Omron CX-Programmer project NewProject (CX-Programmer 9.73)

# PLC NewPLC1: CP1L M

## Global symbols (name address type ; comment)
0.00 BOOL  ; START
0.01 BOOL  ; STOP
0.02 BOOL  ; SOL 2A
0.03 BOOL  ; SOL 2B
0.04 BOOL  ; SOL 3A
0.05 BOOL  ; SOL 4A
0.06 BOOL  ; CONVEYOR
0.07 BOOL  ; RODLESS L
0.08 BOOL  ; RODLESS R
0.10 BOOL  ; GRIPPER CLOSE
0.11 BOOL  ; 3A UP
100.00 BOOL  ; 1A
100.01 BOOL  ; 1B
100.02 BOOL  ; SOL 2A
100.03 BOOL  ; SOL 2B
100.04 BOOL  ; SOL 3A
100.05 BOOL  ; SOL 4A
100.06 BOOL  ; CONVEYOR
1.00 BOOL  ; 3A DOWN
200.00 BOOL  ; TRIGGER
200.01 BOOL  ; 3A UP
200.02 BOOL  ; 3A DOWN
200.03 BOOL  ; 4A OPEN
200.04 BOOL  ; RESET 3A
200.05 BOOL  ; OFF 1B ON 1A
200.06 BOOL  ; RESET
200.07 BOOL  ; RELAY2
200.10 BOOL  ; RELAY3
200.11 BOOL  ; RELAY4
300.00 BOOL  ; RELAY1

## Program UT2 (cyclic task 0)

### Section Section1

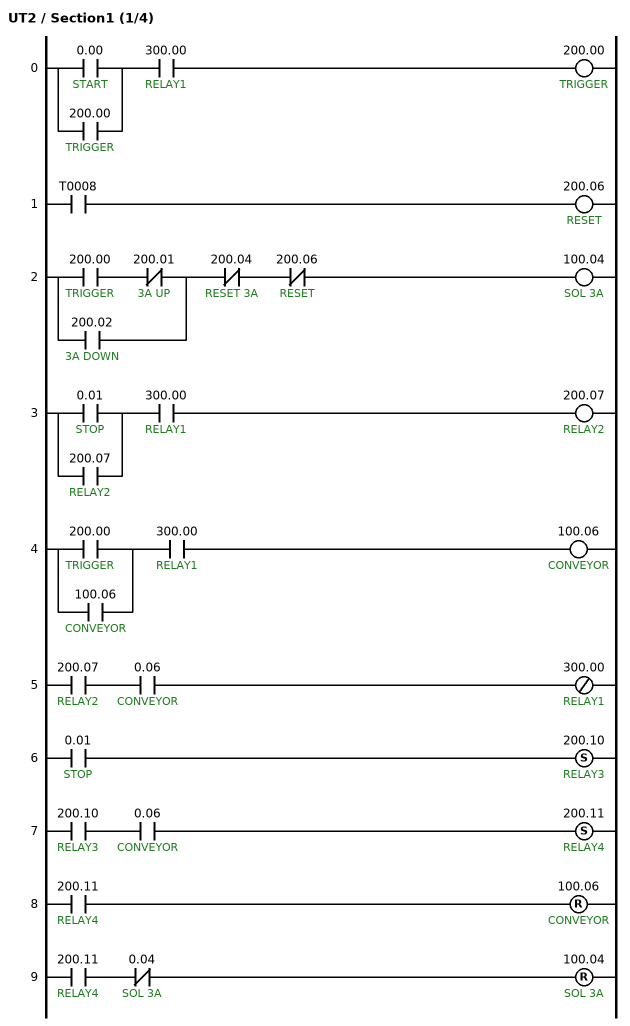
; rung 0
LD 0.00  ; START
OR 200.00  ; TRIGGER
AND 300.00  ; RELAY1
OUT 200.00  ; TRIGGER
; rung 1
LD T0008
OUT 200.06  ; RESET
; rung 2
LD 200.00  ; TRIGGER
ANDNOT 200.01  ; 3A UP
OR 200.02  ; 3A DOWN
ANDNOT 200.04  ; RESET 3A
ANDNOT 200.06  ; RESET
OUT 100.04  ; SOL 3A
; rung 3
LD 0.01  ; STOP
OR 200.07  ; RELAY2
AND 300.00  ; RELAY1
OUT 200.07  ; RELAY2
; rung 4
LD 200.00  ; TRIGGER
OR 100.06  ; CONVEYOR
AND 300.00  ; RELAY1
OUT 100.06  ; CONVEYOR
; rung 5
LD 200.07  ; RELAY2
AND 0.06  ; CONVEYOR
OUTNOT 300.00  ; RELAY1
; rung 6
LD 0.01  ; STOP
SET 200.10  ; RELAY3
; rung 7
LD 200.10  ; RELAY3
AND 0.06  ; CONVEYOR
SET 200.11  ; RELAY4
; rung 8
LD 200.11  ; RELAY4
RSET 100.06  ; CONVEYOR
; rung 9
LD 200.11  ; RELAY4
ANDNOT 0.04  ; SOL 3A
RSET 100.04  ; SOL 3A

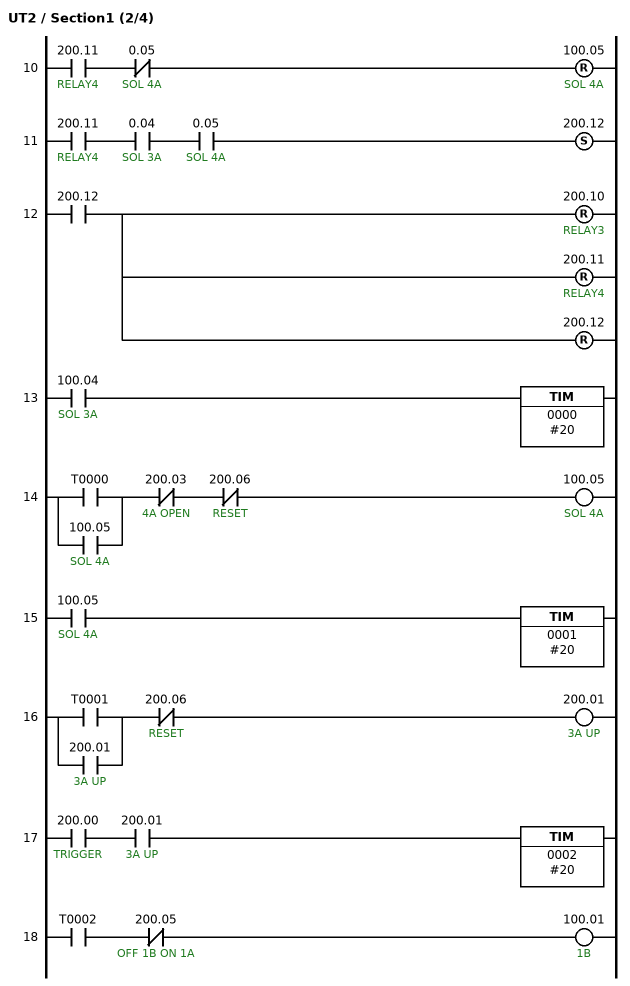
; rung 10
LD 200.11  ; RELAY4
ANDNOT 0.05  ; SOL 4A
RSET 100.05  ; SOL 4A
; rung 11
LD 200.11  ; RELAY4
AND 0.04  ; SOL 3A
AND 0.05  ; SOL 4A
SET 200.12
; rung 12
LD 200.12
RSET 200.10  ; RELAY3
RSET 200.11  ; RELAY4
RSET 200.12
; rung 13
LD 100.04  ; SOL 3A
TIM 0000 #20
; rung 14
LD T0000
OR 100.05  ; SOL 4A
ANDNOT 200.03  ; 4A OPEN
ANDNOT 200.06  ; RESET
OUT 100.05  ; SOL 4A
; rung 15
LD 100.05  ; SOL 4A
TIM 0001 #20
; rung 16
LD T0001
OR 200.01  ; 3A UP
ANDNOT 200.06  ; RESET
OUT 200.01  ; 3A UP
; rung 17
LD 200.00  ; TRIGGER
AND 200.01  ; 3A UP
TIM 0002 #20
; rung 18
LD T0002
ANDNOT 200.05  ; OFF 1B ON 1A
OUT 100.01  ; 1B

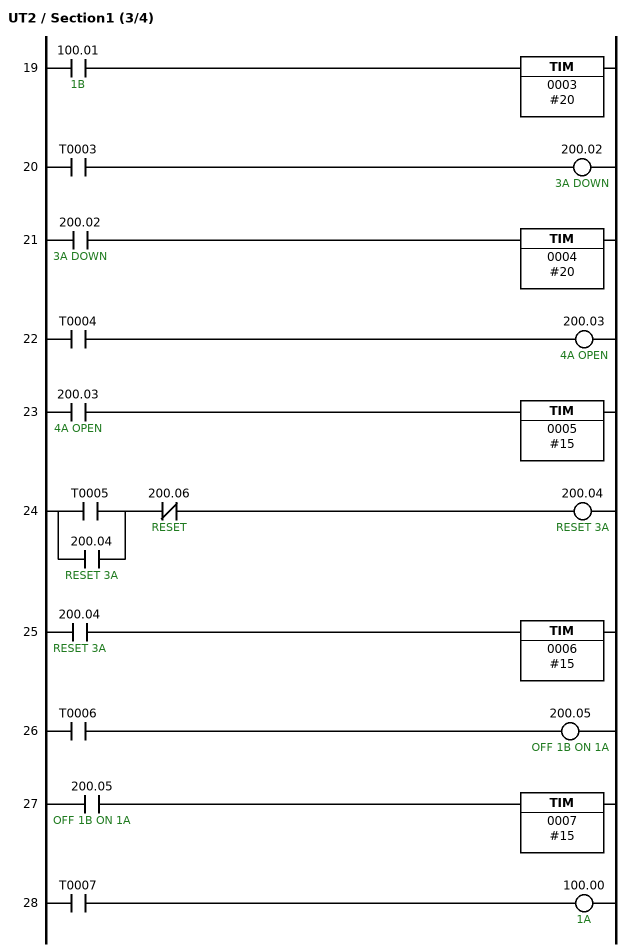
; rung 19
LD 100.01  ; 1B
TIM 0003 #20
; rung 20
LD T0003
OUT 200.02  ; 3A DOWN
; rung 21
LD 200.02  ; 3A DOWN
TIM 0004 #20
; rung 22
LD T0004
OUT 200.03  ; 4A OPEN
; rung 23
LD 200.03  ; 4A OPEN
TIM 0005 #15
; rung 24
LD T0005
OR 200.04  ; RESET 3A
ANDNOT 200.06  ; RESET
OUT 200.04  ; RESET 3A
; rung 25
LD 200.04  ; RESET 3A
TIM 0006 #15
; rung 26
LD T0006
OUT 200.05  ; OFF 1B ON 1A
; rung 27
LD 200.05  ; OFF 1B ON 1A
TIM 0007 #15
; rung 28
LD T0007
OUT 100.00  ; 1A

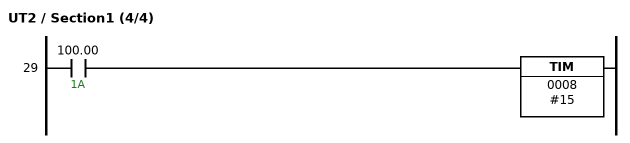
; rung 29
LD 100.00  ; 1A
TIM 0008 #15

### Section END
; rung 0
END(001)